(*
SPDX-FileCopyrightText: © 2026 Oleksandr Tiutyk <trofimich@gmail.com>
SPDX-License-Identifier: MIT
License: https://opensource.org/license/mit
*)

(*!
<summary>Defines a condition for selecting values described by AnyType.</summary>
<description>
A predicate may have configuration and internal state.
Supported data types and treatment of null values are defined by the concrete implementation.
</description>
*)

INTERFACE IPredicate EXTENDS IObject

(*!
<summary>Returns TRUE when the supplied value satisfies this predicate.</summary>
<description>
Must not modify the supplied data or the collection being traversed by the caller.
The predicate may update its own internal state without violating these restrictions.
</description>
*)
//!<param name="valueToCompare">Descriptor of the value to evaluate according to this predicate's supported types and null policy.</param>
METHOD Check : BOOL
VAR_INPUT
	valueToCompare : __SYSTEM.AnyType; 
END_VAR
END_METHOD

END_INTERFACE

(* stored: Version 1.1.0.1
   Itf IPredicate: Id {2d6a38ba-260b-4d26-a5bc-9bd5e6db19e8}
   Method Check: Id {481953a6-7290-46b0-ac08-ad672ed4bf66} *)
